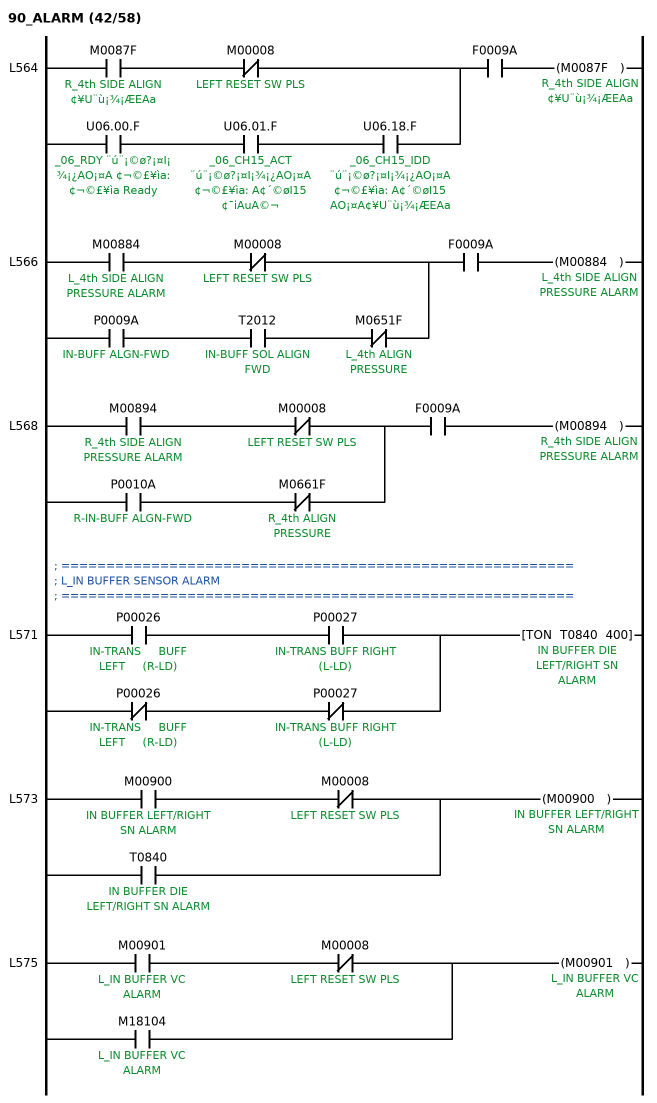
[picture p408: 90_ALARM rungs L564-L575]
; L564
LOAD      M0087F	// R_4th SIDE ALIGN ¢¥U¨ù¡¾¡ÆEAa
AND NOT   M00008	// LEFT RESET SW PLS
LOAD      U06.00.F	// _06_RDY ¨ú¨¡©ø?¡¤I¡¾¡¿AO¡¤A ¢¬©£¥ìa: ¢¬©£¥ìa Ready
AND       U06.01.F	// _06_CH15_ACT ¨ú¨¡©ø?¡¤I¡¾¡¿AO¡¤A ¢¬©£¥ìa: A¢´©øI15 ¢¯iAuA©¬
AND       U06.18.F	// _06_CH15_IDD ¨ú¨¡©ø?¡¤I¡¾¡¿AO¡¤A ¢¬©£¥ìa: A¢´©øI15 AO¡¤A¢¥U¨ù¡¾¡ÆEAa
OR LOAD
AND       F0009A
OUT       M0087F	// R_4th SIDE ALIGN ¢¥U¨ù¡¾¡ÆEAa
; L566
LOAD      M00884	// L_4th SIDE ALIGN PRESSURE ALARM
AND NOT   M00008	// LEFT RESET SW PLS
LOAD      P0009A	// IN-BUFF ALGN-FWD
AND       T2012	// IN-BUFF SOL ALIGN FWD
AND NOT   M0651F	// L_4th ALIGN PRESSURE
OR LOAD
AND       F0009A
OUT       M00884	// L_4th SIDE ALIGN PRESSURE ALARM
; L568
LOAD      M00894	// R_4th SIDE ALIGN PRESSURE ALARM
AND NOT   M00008	// LEFT RESET SW PLS
LOAD      P0010A	// R-IN-BUFF ALGN-FWD
AND NOT   M0661F	// R_4th ALIGN PRESSURE
OR LOAD
AND       F0009A
OUT       M00894	// R_4th SIDE ALIGN PRESSURE ALARM
// =========================================================
// 
//        L_IN BUFFER SENSOR ALARM
// 
// =========================================================
; L571
LOAD      P00026	// IN-TRANS     BUFF     LEFT     (R-LD)
AND       P00027	// IN-TRANS BUFF RIGHT     (L-LD)
LOAD NOT  P00026	// IN-TRANS     BUFF     LEFT     (R-LD)
AND NOT   P00027	// IN-TRANS BUFF RIGHT     (L-LD)
OR LOAD
TON       T0840 400	// IN BUFFER DIE LEFT/RIGHT SN ALARM
; L573
LOAD      M00900	// IN BUFFER LEFT/RIGHT SN ALARM
AND NOT   M00008	// LEFT RESET SW PLS
OR        T0840	// IN BUFFER DIE LEFT/RIGHT SN ALARM
OUT       M00900	// IN BUFFER LEFT/RIGHT SN ALARM
; L575
LOAD      M00901	// L_IN BUFFER VC ALARM
AND NOT   M00008	// LEFT RESET SW PLS
OR        M18104	// L_IN BUFFER VC ALARM
OUT       M00901	// L_IN BUFFER VC ALARM

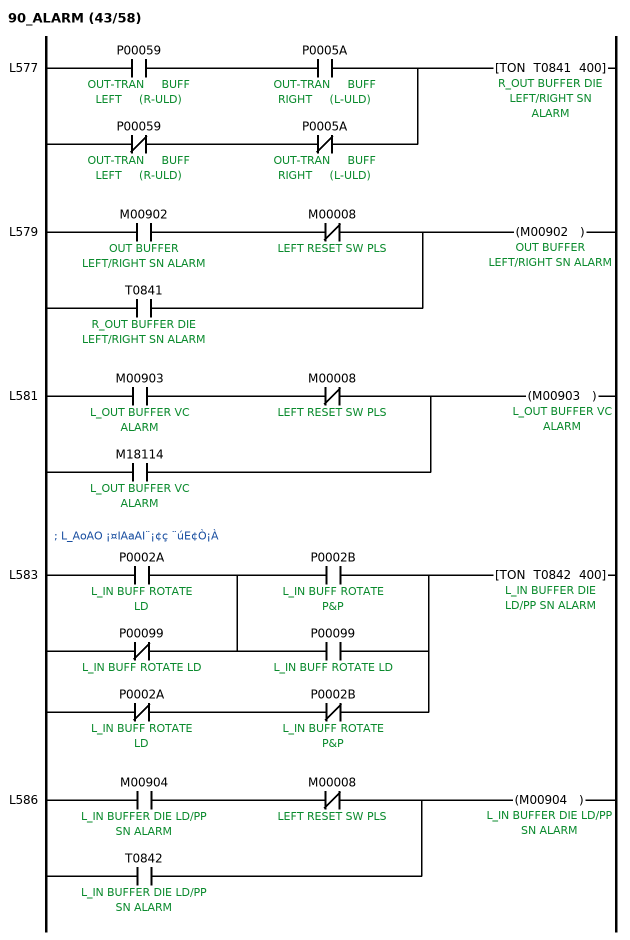
; L577
LOAD      P00059	// OUT-TRAN     BUFF     LEFT     (R-ULD)
AND       P0005A	// OUT-TRAN     BUFF     RIGHT     (L-ULD)
LOAD NOT  P00059	// OUT-TRAN     BUFF     LEFT     (R-ULD)
AND NOT   P0005A	// OUT-TRAN     BUFF     RIGHT     (L-ULD)
OR LOAD
TON       T0841 400	// R_OUT BUFFER DIE LEFT/RIGHT SN ALARM
; L579
LOAD      M00902	// OUT BUFFER LEFT/RIGHT SN ALARM
AND NOT   M00008	// LEFT RESET SW PLS
OR        T0841	// R_OUT BUFFER DIE LEFT/RIGHT SN ALARM
OUT       M00902	// OUT BUFFER LEFT/RIGHT SN ALARM
; L581
LOAD      M00903	// L_OUT BUFFER VC ALARM
AND NOT   M00008	// LEFT RESET SW PLS
OR        M18114	// L_OUT BUFFER VC ALARM
OUT       M00903	// L_OUT BUFFER VC ALARM
; L583
LOAD      P0002A	// L_IN BUFF ROTATE     LD
OR NOT    P00099	// L_IN BUFF ROTATE LD
LOAD      P0002B	// L_IN BUFF ROTATE      P&P
OR        P00099	// L_IN BUFF ROTATE LD
AND LOAD
LOAD NOT  P0002A	// L_IN BUFF ROTATE     LD
AND NOT   P0002B	// L_IN BUFF ROTATE      P&P
OR LOAD
TON       T0842 400	// L_IN BUFFER DIE LD/PP SN ALARM
// output comment: L_AoAO ¡¤IAaAI¨¡¢ç ¨úE¢Ò¡À
; L586
LOAD      M00904	// L_IN BUFFER DIE LD/PP SN ALARM
AND NOT   M00008	// LEFT RESET SW PLS
OR        T0842	// L_IN BUFFER DIE LD/PP SN ALARM
OUT       M00904	// L_IN BUFFER DIE LD/PP SN ALARM

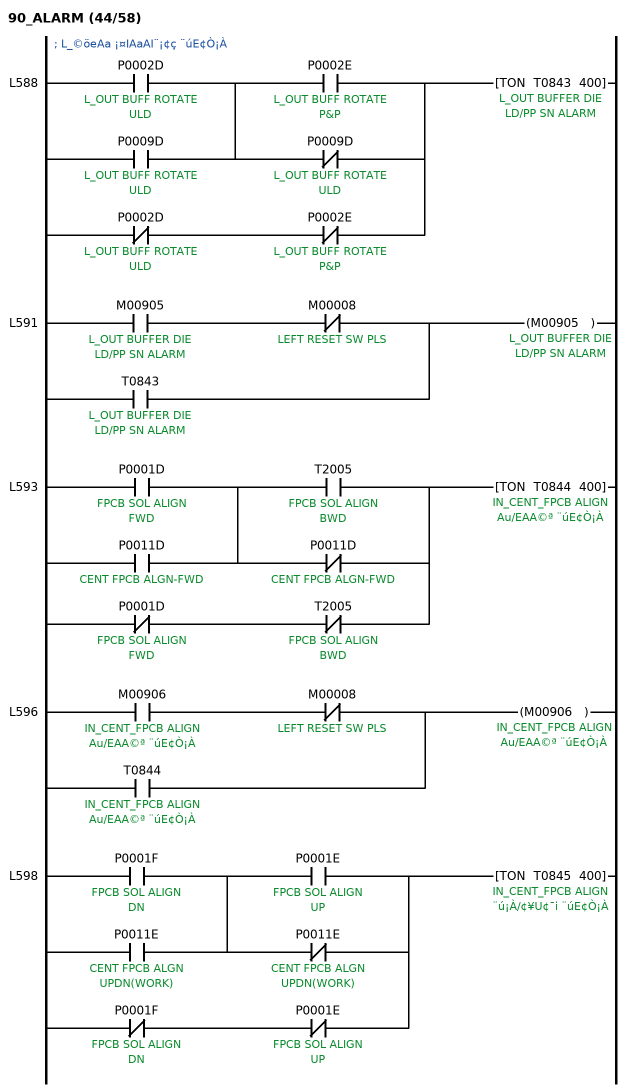
; L588
LOAD      P0002D	// L_OUT BUFF ROTATE     ULD
OR        P0009D	// L_OUT BUFF ROTATE ULD
LOAD      P0002E	// L_OUT BUFF ROTATE      P&P
OR NOT    P0009D	// L_OUT BUFF ROTATE ULD
AND LOAD
LOAD NOT  P0002D	// L_OUT BUFF ROTATE     ULD
AND NOT   P0002E	// L_OUT BUFF ROTATE      P&P
OR LOAD
TON       T0843 400	// L_OUT BUFFER DIE LD/PP SN ALARM
// output comment: L_©öeAa ¡¤IAaAI¨¡¢ç ¨úE¢Ò¡À
; L591
LOAD      M00905	// L_OUT BUFFER DIE LD/PP SN ALARM
AND NOT   M00008	// LEFT RESET SW PLS
OR        T0843	// L_OUT BUFFER DIE LD/PP SN ALARM
OUT       M00905	// L_OUT BUFFER DIE LD/PP SN ALARM
; L593
LOAD      P0001D	// FPCB SOL ALIGN         FWD
OR        P0011D	// CENT FPCB ALGN-FWD
LOAD      T2005	// FPCB SOL ALIGN         BWD
OR NOT    P0011D	// CENT FPCB ALGN-FWD
AND LOAD
LOAD NOT  P0001D	// FPCB SOL ALIGN         FWD
AND NOT   T2005	// FPCB SOL ALIGN         BWD
OR LOAD
TON       T0844 400	// IN_CENT_FPCB ALIGN Au/EAA©ª ¨úE¢Ò¡À
; L596
LOAD      M00906	// IN_CENT_FPCB ALIGN Au/EAA©ª ¨úE¢Ò¡À
AND NOT   M00008	// LEFT RESET SW PLS
OR        T0844	// IN_CENT_FPCB ALIGN Au/EAA©ª ¨úE¢Ò¡À
OUT       M00906	// IN_CENT_FPCB ALIGN Au/EAA©ª ¨úE¢Ò¡À
; L598
LOAD      P0001F	// FPCB SOL ALIGN        DN
OR        P0011E	// CENT FPCB ALGN UPDN(WORK)
LOAD      P0001E	// FPCB SOL ALIGN         UP
OR NOT    P0011E	// CENT FPCB ALGN UPDN(WORK)
AND LOAD
LOAD NOT  P0001F	// FPCB SOL ALIGN        DN
AND NOT   P0001E	// FPCB SOL ALIGN         UP
OR LOAD
TON       T0845 400	// IN_CENT_FPCB ALIGN ¨ú¡À/¢¥U¢¯i ¨úE¢Ò¡À

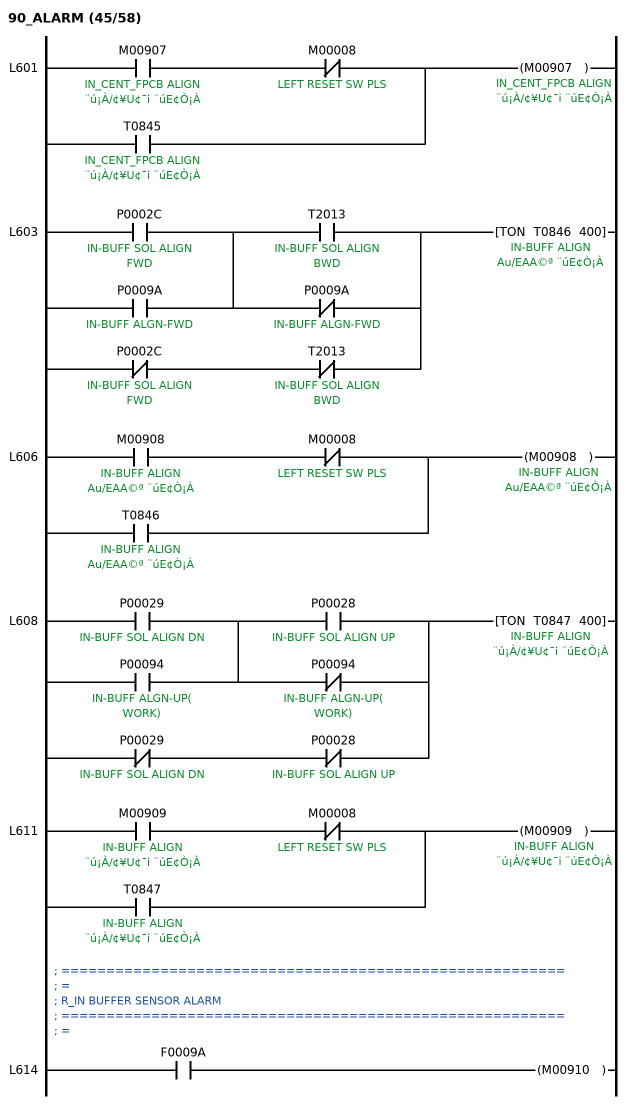
; L601
LOAD      M00907	// IN_CENT_FPCB ALIGN ¨ú¡À/¢¥U¢¯i ¨úE¢Ò¡À
AND NOT   M00008	// LEFT RESET SW PLS
OR        T0845	// IN_CENT_FPCB ALIGN ¨ú¡À/¢¥U¢¯i ¨úE¢Ò¡À
OUT       M00907	// IN_CENT_FPCB ALIGN ¨ú¡À/¢¥U¢¯i ¨úE¢Ò¡À
; L603
LOAD      P0002C	// IN-BUFF SOL ALIGN FWD
OR        P0009A	// IN-BUFF ALGN-FWD
LOAD      T2013	// IN-BUFF SOL ALIGN BWD
OR NOT    P0009A	// IN-BUFF ALGN-FWD
AND LOAD
LOAD NOT  P0002C	// IN-BUFF SOL ALIGN FWD
AND NOT   T2013	// IN-BUFF SOL ALIGN BWD
OR LOAD
TON       T0846 400	// IN-BUFF ALIGN Au/EAA©ª ¨úE¢Ò¡À
; L606
LOAD      M00908	// IN-BUFF ALIGN Au/EAA©ª ¨úE¢Ò¡À
AND NOT   M00008	// LEFT RESET SW PLS
OR        T0846	// IN-BUFF ALIGN Au/EAA©ª ¨úE¢Ò¡À
OUT       M00908	// IN-BUFF ALIGN Au/EAA©ª ¨úE¢Ò¡À
; L608
LOAD      P00029	// IN-BUFF SOL ALIGN DN
OR        P00094	// IN-BUFF ALGN-UP(WORK)
LOAD      P00028	// IN-BUFF SOL ALIGN UP
OR NOT    P00094	// IN-BUFF ALGN-UP(WORK)
AND LOAD
LOAD NOT  P00029	// IN-BUFF SOL ALIGN DN
AND NOT   P00028	// IN-BUFF SOL ALIGN UP
OR LOAD
TON       T0847 400	// IN-BUFF ALIGN ¨ú¡À/¢¥U¢¯i ¨úE¢Ò¡À
; L611
LOAD      M00909	// IN-BUFF ALIGN ¨ú¡À/¢¥U¢¯i ¨úE¢Ò¡À
AND NOT   M00008	// LEFT RESET SW PLS
OR        T0847	// IN-BUFF ALIGN ¨ú¡À/¢¥U¢¯i ¨úE¢Ò¡À
OUT       M00909	// IN-BUFF ALIGN ¨ú¡À/¢¥U¢¯i ¨úE¢Ò¡À
// =========================================================
// 
//        R_IN BUFFER SENSOR ALARM
// 
// =========================================================
; L614
LOAD      F0009A
OUT       M00910

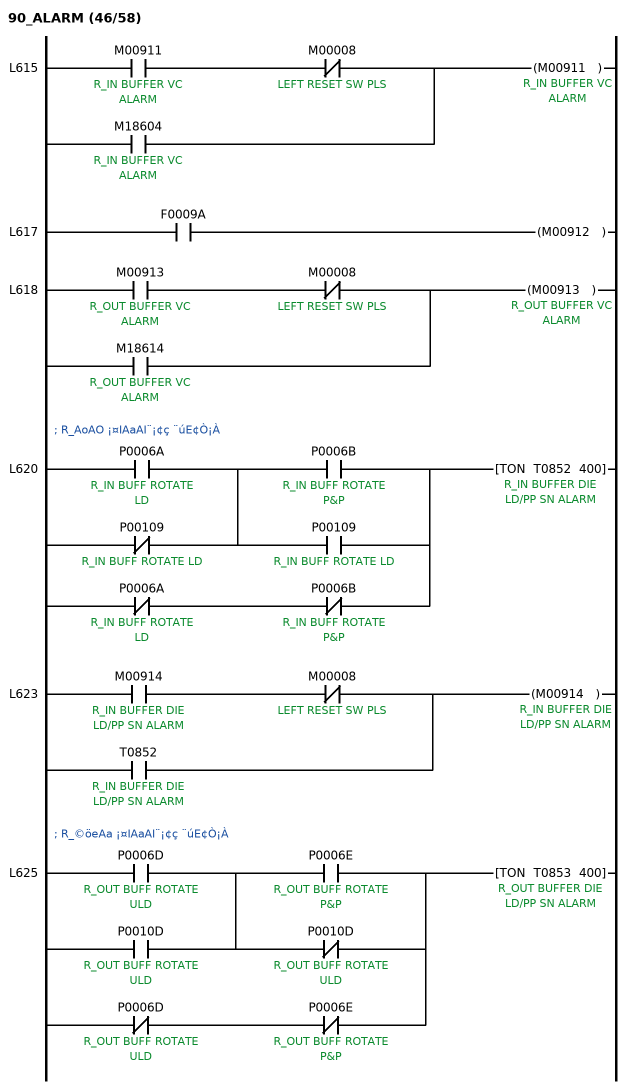
; L615
LOAD      M00911	// R_IN BUFFER VC ALARM
AND NOT   M00008	// LEFT RESET SW PLS
OR        M18604	// R_IN BUFFER VC ALARM
OUT       M00911	// R_IN BUFFER VC ALARM
; L617
LOAD      F0009A
OUT       M00912
; L618
LOAD      M00913	// R_OUT BUFFER VC ALARM
AND NOT   M00008	// LEFT RESET SW PLS
OR        M18614	// R_OUT BUFFER VC ALARM
OUT       M00913	// R_OUT BUFFER VC ALARM
; L620
LOAD      P0006A	// R_IN BUFF ROTATE      LD
OR NOT    P00109	// R_IN BUFF ROTATE LD
LOAD      P0006B	// R_IN BUFF ROTATE      P&P
OR        P00109	// R_IN BUFF ROTATE LD
AND LOAD
LOAD NOT  P0006A	// R_IN BUFF ROTATE      LD
AND NOT   P0006B	// R_IN BUFF ROTATE      P&P
OR LOAD
TON       T0852 400	// R_IN BUFFER DIE LD/PP SN ALARM
// output comment: R_AoAO ¡¤IAaAI¨¡¢ç ¨úE¢Ò¡À
; L623
LOAD      M00914	// R_IN BUFFER DIE LD/PP SN ALARM
AND NOT   M00008	// LEFT RESET SW PLS
OR        T0852	// R_IN BUFFER DIE LD/PP SN ALARM
OUT       M00914	// R_IN BUFFER DIE LD/PP SN ALARM
; L625
LOAD      P0006D	// R_OUT BUFF ROTATE      ULD
OR        P0010D	// R_OUT BUFF ROTATE ULD
LOAD      P0006E	// R_OUT BUFF ROTATE      P&P
OR NOT    P0010D	// R_OUT BUFF ROTATE ULD
AND LOAD
LOAD NOT  P0006D	// R_OUT BUFF ROTATE      ULD
AND NOT   P0006E	// R_OUT BUFF ROTATE      P&P
OR LOAD
TON       T0853 400	// R_OUT BUFFER DIE LD/PP SN ALARM
// output comment: R_©öeAa ¡¤IAaAI¨¡¢ç ¨úE¢Ò¡À

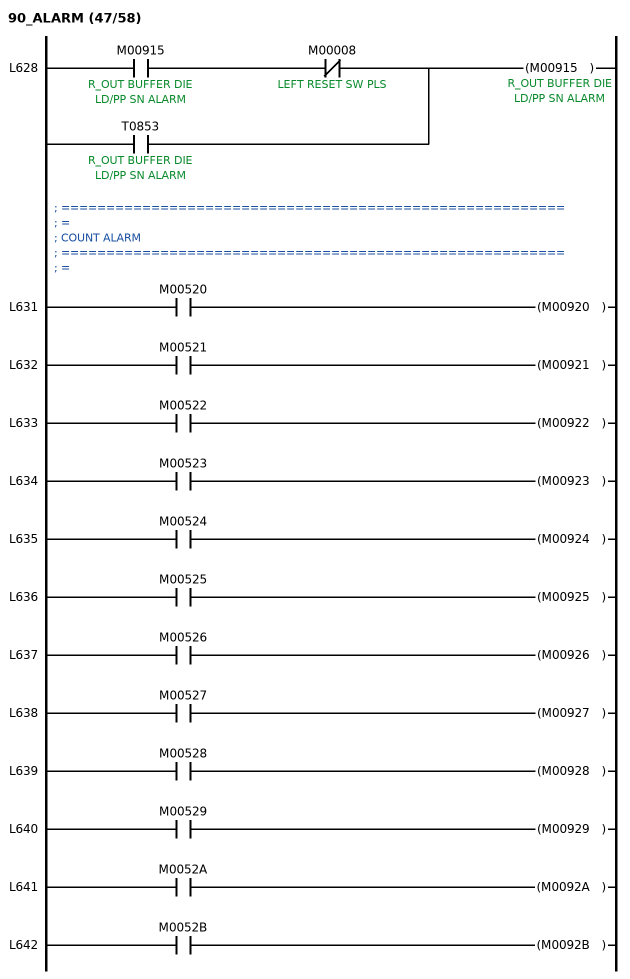
; L628
LOAD      M00915	// R_OUT BUFFER DIE LD/PP SN ALARM
AND NOT   M00008	// LEFT RESET SW PLS
OR        T0853	// R_OUT BUFFER DIE LD/PP SN ALARM
OUT       M00915	// R_OUT BUFFER DIE LD/PP SN ALARM
// =========================================================
// 
//       COUNT ALARM
// 
// =========================================================
; L631
LOAD      M00520
OUT       M00920
; L632
LOAD      M00521
OUT       M00921
; L633
LOAD      M00522
OUT       M00922
; L634
LOAD      M00523
OUT       M00923
; L635
LOAD      M00524
OUT       M00924
; L636
LOAD      M00525
OUT       M00925
; L637
LOAD      M00526
OUT       M00926
; L638
LOAD      M00527
OUT       M00927
; L639
LOAD      M00528
OUT       M00928
; L640
LOAD      M00529
OUT       M00929
; L641
LOAD      M0052A
OUT       M0092A
; L642
LOAD      M0052B
OUT       M0092B

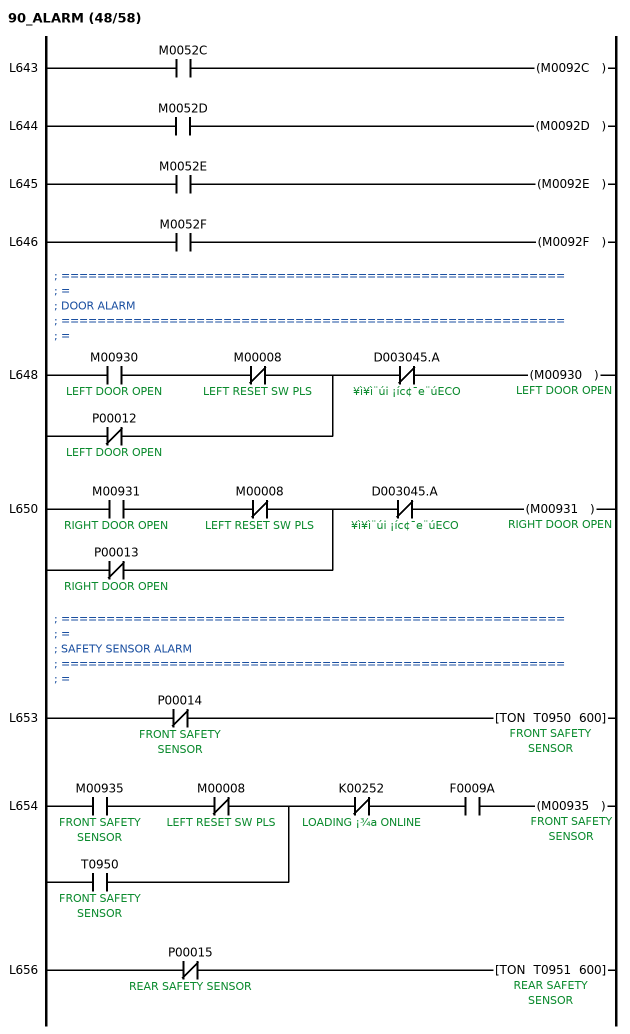
; L643
LOAD      M0052C
OUT       M0092C
; L644
LOAD      M0052D
OUT       M0092D
; L645
LOAD      M0052E
OUT       M0092E
; L646
LOAD      M0052F
OUT       M0092F
// =========================================================
// 
//       DOOR ALARM
// 
// =========================================================
; L648
LOAD      M00930	// LEFT DOOR OPEN
AND NOT   M00008	// LEFT RESET SW PLS
OR NOT    P00012	// LEFT DOOR OPEN
AND NOT   D003045.A	// ¥ì¥ì¨úi ¡íc¢¯e¨úECO
OUT       M00930	// LEFT DOOR OPEN
; L650
LOAD      M00931	// RIGHT DOOR OPEN
AND NOT   M00008	// LEFT RESET SW PLS
OR NOT    P00013	// RIGHT DOOR OPEN
AND NOT   D003045.A	// ¥ì¥ì¨úi ¡íc¢¯e¨úECO
OUT       M00931	// RIGHT DOOR OPEN
// =========================================================
// 
//       SAFETY SENSOR ALARM
// 
// =========================================================
; L653
LOAD NOT  P00014	// FRONT SAFETY SENSOR
TON       T0950 600	// FRONT SAFETY SENSOR
; L654
LOAD      M00935	// FRONT SAFETY SENSOR
AND NOT   M00008	// LEFT RESET SW PLS
OR        T0950	// FRONT SAFETY SENSOR
AND NOT   K00252	// LOADING ¡¾a ONLINE
AND       F0009A
OUT       M00935	// FRONT SAFETY SENSOR
; L656
LOAD NOT  P00015	// REAR SAFETY SENSOR
TON       T0951 600	// REAR SAFETY SENSOR

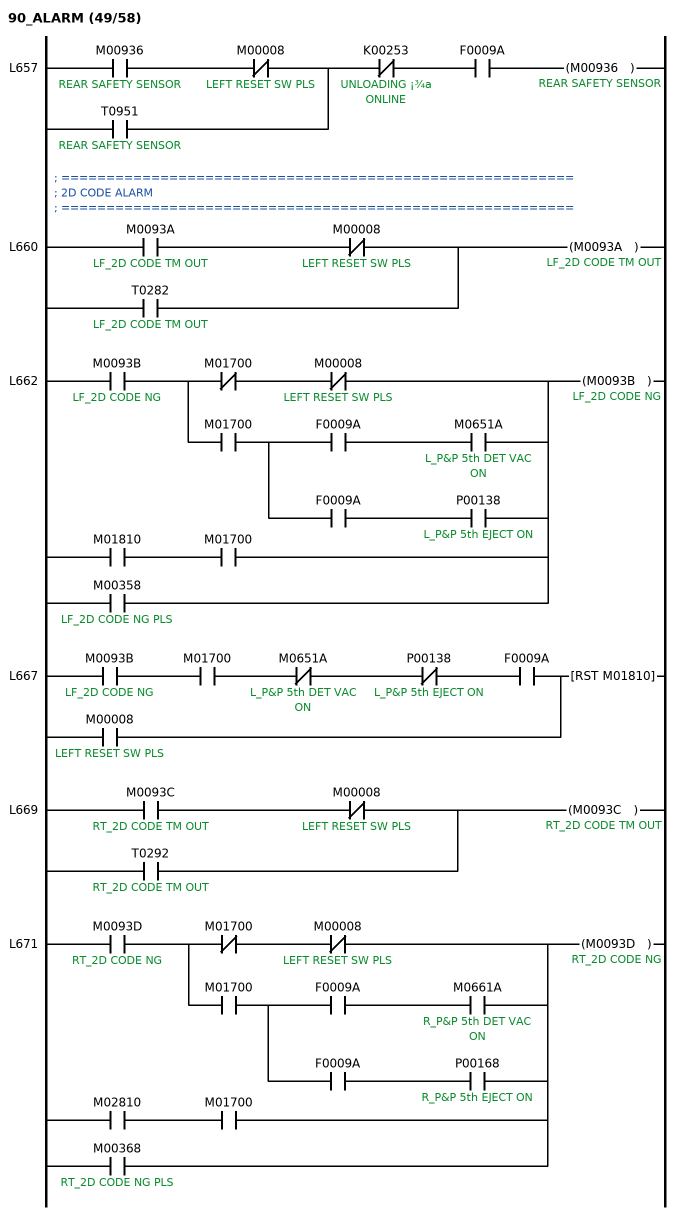
; L657
LOAD      M00936	// REAR SAFETY SENSOR
AND NOT   M00008	// LEFT RESET SW PLS
OR        T0951	// REAR SAFETY SENSOR
AND NOT   K00253	// UNLOADING ¡¾a ONLINE
AND       F0009A
OUT       M00936	// REAR SAFETY SENSOR
// =========================================================
// 
//       2D CODE ALARM
// 
// =========================================================
; L660
LOAD      M0093A	// LF_2D CODE TM OUT
AND NOT   M00008	// LEFT RESET SW PLS
OR        T0282	// LF_2D CODE TM OUT
OUT       M0093A	// LF_2D CODE TM OUT
; L662
LOAD      M0093B	// LF_2D CODE NG
LOAD NOT  M01700
AND NOT   M00008	// LEFT RESET SW PLS
LOAD      M01700
LOAD      F0009A
AND       M0651A	// L_P&P 5th DET VAC ON
LOAD      F0009A
AND       P00138	// L_P&P 5th EJECT ON
OR LOAD
AND LOAD
OR LOAD
AND LOAD
LOAD      M01810
AND       M01700
OR LOAD
OR        M00358	// LF_2D CODE NG PLS
OUT       M0093B	// LF_2D CODE NG
; L667
LOAD      M0093B	// LF_2D CODE NG
AND       M01700
AND NOT   M0651A	// L_P&P 5th DET VAC ON
AND NOT   P00138	// L_P&P 5th EJECT ON
AND       F0009A
OR        M00008	// LEFT RESET SW PLS
RST       M01810
; L669
LOAD      M0093C	// RT_2D CODE TM OUT
AND NOT   M00008	// LEFT RESET SW PLS
OR        T0292	// RT_2D CODE TM OUT
OUT       M0093C	// RT_2D CODE TM OUT
; L671
LOAD      M0093D	// RT_2D CODE NG
LOAD NOT  M01700
AND NOT   M00008	// LEFT RESET SW PLS
LOAD      M01700
LOAD      F0009A
AND       M0661A	// R_P&P 5th DET VAC ON
LOAD      F0009A
AND       P00168	// R_P&P 5th EJECT ON
OR LOAD
AND LOAD
OR LOAD
AND LOAD
LOAD      M02810
AND       M01700
OR LOAD
OR        M00368	// RT_2D CODE NG PLS
OUT       M0093D	// RT_2D CODE NG

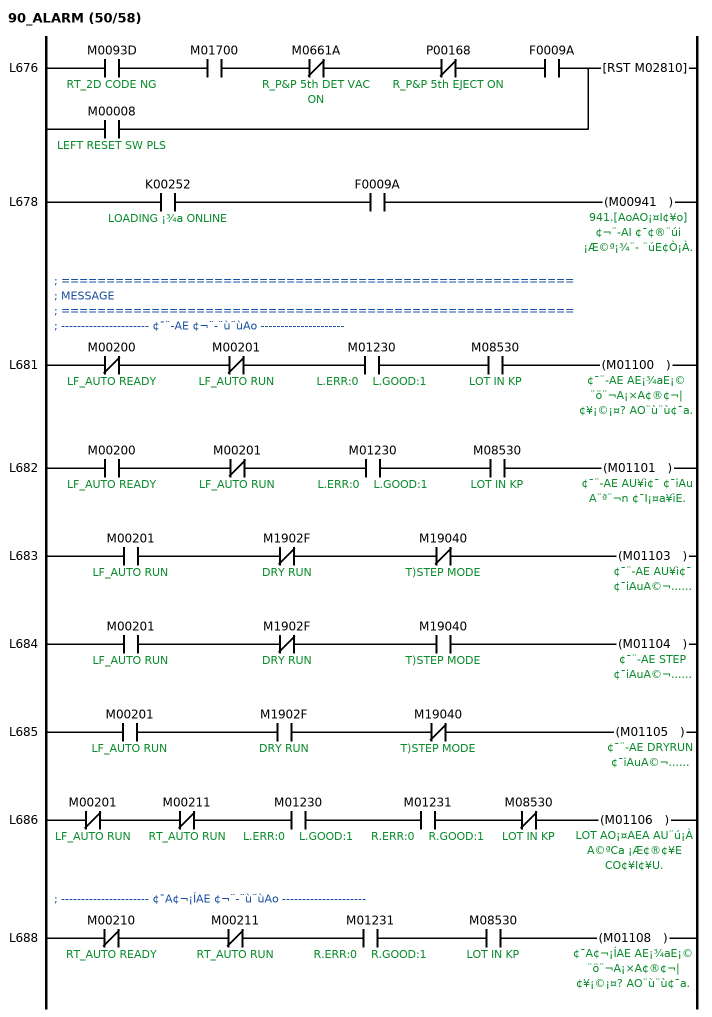
; L676
LOAD      M0093D	// RT_2D CODE NG
AND       M01700
AND NOT   M0661A	// R_P&P 5th DET VAC ON
AND NOT   P00168	// R_P&P 5th EJECT ON
AND       F0009A
OR        M00008	// LEFT RESET SW PLS
RST       M02810
; L678
LOAD      K00252	// LOADING ¡¾a ONLINE
AND       F0009A
OUT       M00941	// 941.[AoAO¡¤I¢¥o] ¢¬¨­AI ¢¯¢®¨úi ¡Æ©ª¡¾¨­ ¨úE¢Ò¡À.
// =========================================================
// 
//       MESSAGE
// 
// =========================================================
// ---------------------- ¢¯¨­AE ¢¬¨­¨ù¨ùAo ---------------------
; L681
LOAD NOT  M00200	// LF_AUTO READY
AND NOT   M00201	// LF_AUTO RUN
AND       M01230	// L.ERR:0    L.GOOD:1
AND       M08530	// LOT IN KP
OUT       M01100	// ¢¯¨­AE AE¡¾aE¡© ¨ö¨¬A¡×A¢®¢¬| ¢¥¡©¡¤? AO¨ù¨ù¢¯a.
; L682
LOAD      M00200	// LF_AUTO READY
AND NOT   M00201	// LF_AUTO RUN
AND       M01230	// L.ERR:0    L.GOOD:1
AND       M08530	// LOT IN KP
OUT       M01101	// ¢¯¨­AE AU¥ì¢¯ ¢¯iAu A¨ª¨¬n ¢¯I¡¤a¥ìE.
; L683
LOAD      M00201	// LF_AUTO RUN
AND NOT   M1902F	// DRY RUN
AND NOT   M19040	// T)STEP MODE
OUT       M01103	// ¢¯¨­AE AU¥ì¢¯ ¢¯iAuA©¬......
; L684
LOAD      M00201	// LF_AUTO RUN
AND NOT   M1902F	// DRY RUN
AND       M19040	// T)STEP MODE
OUT       M01104	// ¢¯¨­AE STEP ¢¯iAuA©¬......
; L685
LOAD      M00201	// LF_AUTO RUN
AND       M1902F	// DRY RUN
AND NOT   M19040	// T)STEP MODE
OUT       M01105	// ¢¯¨­AE DRYRUN ¢¯iAuA©¬......
; L686
LOAD NOT  M00201	// LF_AUTO RUN
AND NOT   M00211	// RT_AUTO RUN
AND       M01230	// L.ERR:0    L.GOOD:1
AND       M01231	// R.ERR:0    R.GOOD:1
AND NOT   M08530	// LOT IN KP
OUT       M01106	// LOT AO¡¤AEA AU¨ú¡À A©ªCa ¡Æ¢®¢¥E CO¢¥I¢¥U.
// ---------------------- ¢¯A¢¬¡ÍAE ¢¬¨­¨ù¨ùAo ---------------------
; L688
LOAD NOT  M00210	// RT_AUTO READY
AND NOT   M00211	// RT_AUTO RUN
AND       M01231	// R.ERR:0    R.GOOD:1
AND       M08530	// LOT IN KP
OUT       M01108	// ¢¯A¢¬¡ÍAE AE¡¾aE¡© ¨ö¨¬A¡×A¢®¢¬| ¢¥¡©¡¤? AO¨ù¨ù¢¯a.

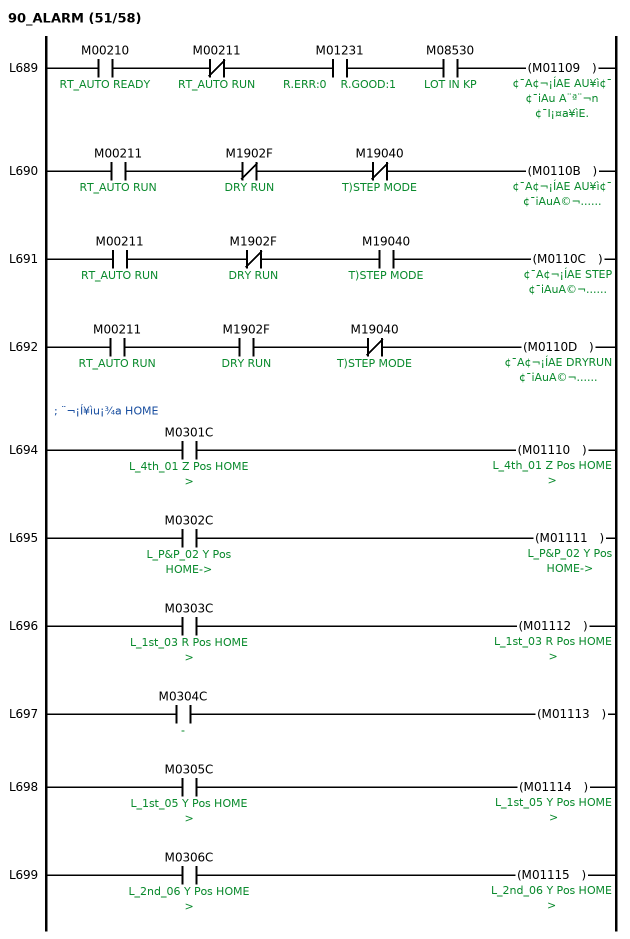
; L689
LOAD      M00210	// RT_AUTO READY
AND NOT   M00211	// RT_AUTO RUN
AND       M01231	// R.ERR:0    R.GOOD:1
AND       M08530	// LOT IN KP
OUT       M01109	// ¢¯A¢¬¡ÍAE AU¥ì¢¯ ¢¯iAu A¨ª¨¬n ¢¯I¡¤a¥ìE.
; L690
LOAD      M00211	// RT_AUTO RUN
AND NOT   M1902F	// DRY RUN
AND NOT   M19040	// T)STEP MODE
OUT       M0110B	// ¢¯A¢¬¡ÍAE AU¥ì¢¯ ¢¯iAuA©¬......
; L691
LOAD      M00211	// RT_AUTO RUN
AND NOT   M1902F	// DRY RUN
AND       M19040	// T)STEP MODE
OUT       M0110C	// ¢¯A¢¬¡ÍAE STEP ¢¯iAuA©¬......
; L692
LOAD      M00211	// RT_AUTO RUN
AND       M1902F	// DRY RUN
AND NOT   M19040	// T)STEP MODE
OUT       M0110D	// ¢¯A¢¬¡ÍAE DRYRUN ¢¯iAuA©¬......
// ¨¬¡Í¥ìu¡¾a HOME
; L694
LOAD      M0301C	// L_4th_01 Z Pos HOME >
OUT       M01110	// L_4th_01 Z Pos HOME >
; L695
LOAD      M0302C	// L_P&P_02 Y Pos HOME->
OUT       M01111	// L_P&P_02 Y Pos HOME->
; L696
LOAD      M0303C	// L_1st_03 R Pos HOME >
OUT       M01112	// L_1st_03 R Pos HOME >
; L697
LOAD      M0304C	// -
OUT       M01113
; L698
LOAD      M0305C	// L_1st_05 Y Pos HOME >
OUT       M01114	// L_1st_05 Y Pos HOME >
; L699
LOAD      M0306C	// L_2nd_06 Y Pos HOME >
OUT       M01115	// L_2nd_06 Y Pos HOME >

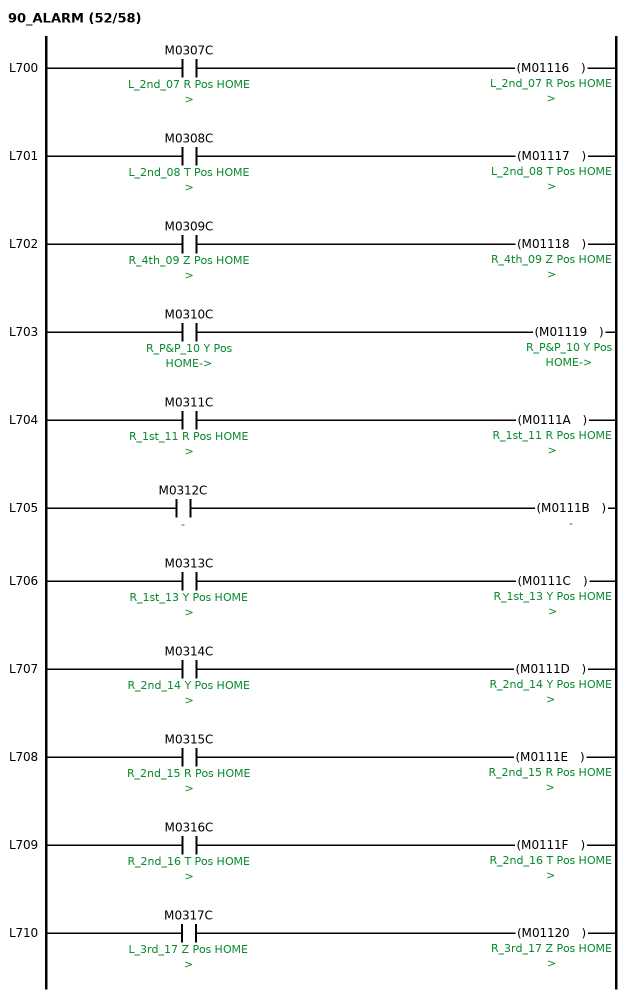
; L700
LOAD      M0307C	// L_2nd_07 R Pos HOME >
OUT       M01116	// L_2nd_07 R Pos HOME >
; L701
LOAD      M0308C	// L_2nd_08 T Pos HOME >
OUT       M01117	// L_2nd_08 T Pos HOME >
; L702
LOAD      M0309C	// R_4th_09 Z Pos HOME >
OUT       M01118	// R_4th_09 Z Pos HOME >
; L703
LOAD      M0310C	// R_P&P_10 Y Pos HOME->
OUT       M01119	// R_P&P_10 Y Pos HOME->
; L704
LOAD      M0311C	// R_1st_11 R Pos HOME >
OUT       M0111A	// R_1st_11 R Pos HOME >
; L705
LOAD      M0312C	// -
OUT       M0111B	// -
; L706
LOAD      M0313C	// R_1st_13 Y Pos HOME >
OUT       M0111C	// R_1st_13 Y Pos HOME >
; L707
LOAD      M0314C	// R_2nd_14 Y Pos HOME >
OUT       M0111D	// R_2nd_14 Y Pos HOME >
; L708
LOAD      M0315C	// R_2nd_15 R Pos HOME >
OUT       M0111E	// R_2nd_15 R Pos HOME >
; L709
LOAD      M0316C	// R_2nd_16 T Pos HOME >
OUT       M0111F	// R_2nd_16 T Pos HOME >
; L710
LOAD      M0317C	// L_3rd_17 Z Pos HOME >
OUT       M01120	// R_3rd_17 Z Pos HOME >

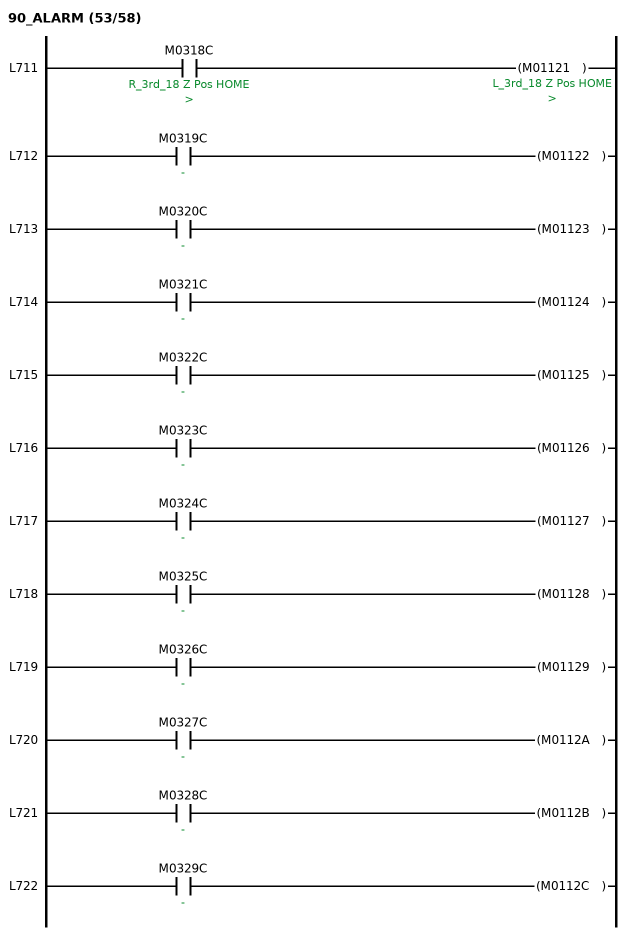
; L711
LOAD      M0318C	// R_3rd_18 Z Pos HOME >
OUT       M01121	// L_3rd_18 Z Pos HOME >
; L712
LOAD      M0319C	// -
OUT       M01122
; L713
LOAD      M0320C	// -
OUT       M01123
; L714
LOAD      M0321C	// -
OUT       M01124
; L715
LOAD      M0322C	// -
OUT       M01125
; L716
LOAD      M0323C	// -
OUT       M01126
; L717
LOAD      M0324C	// -
OUT       M01127
; L718
LOAD      M0325C	// -
OUT       M01128
; L719
LOAD      M0326C	// -
OUT       M01129
; L720
LOAD      M0327C	// -
OUT       M0112A
; L721
LOAD      M0328C	// -
OUT       M0112B
; L722
LOAD      M0329C	// -
OUT       M0112C

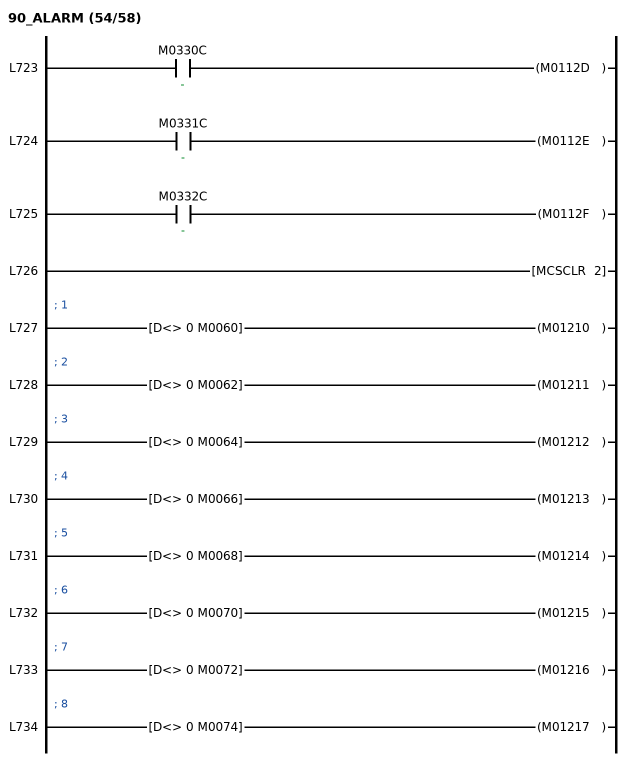
; L723
LOAD      M0330C	// -
OUT       M0112D
; L724
LOAD      M0331C	// -
OUT       M0112E
; L725
LOAD      M0332C	// -
OUT       M0112F
; L726
MCSCLR    2
; L727
LOADD<>   0 M0060
OUT       M01210
// output comment: 1
; L728
LOADD<>   0 M0062
OUT       M01211
// output comment: 2
; L729
LOADD<>   0 M0064
OUT       M01212
// output comment: 3
; L730
LOADD<>   0 M0066
OUT       M01213
// output comment: 4
; L731
LOADD<>   0 M0068
OUT       M01214
// output comment: 5
; L732
LOADD<>   0 M0070
OUT       M01215
// output comment: 6
; L733
LOADD<>   0 M0072
OUT       M01216
// output comment: 7
; L734
LOADD<>   0 M0074
OUT       M01217
// output comment: 8

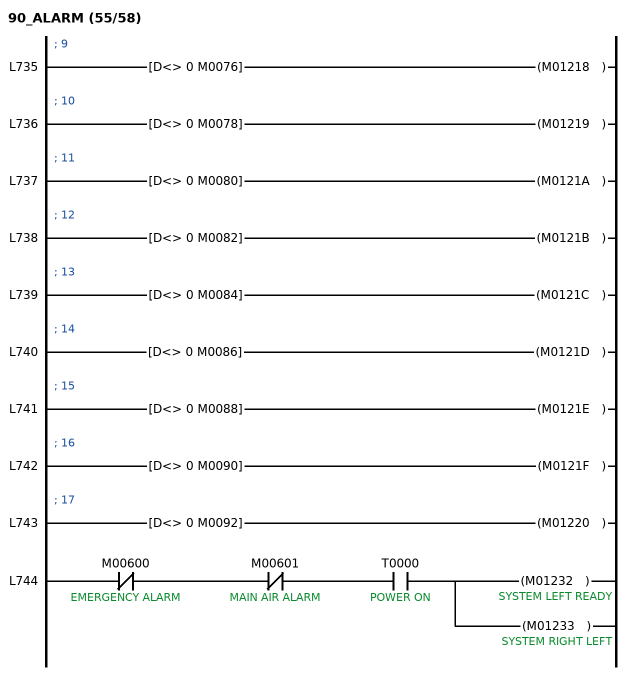
; L735
LOADD<>   0 M0076
OUT       M01218
// output comment: 9
; L736
LOADD<>   0 M0078
OUT       M01219
// output comment: 10
; L737
LOADD<>   0 M0080
OUT       M0121A
// output comment: 11
; L738
LOADD<>   0 M0082
OUT       M0121B
// output comment: 12
; L739
LOADD<>   0 M0084
OUT       M0121C
// output comment: 13
; L740
LOADD<>   0 M0086
OUT       M0121D
// output comment: 14
; L741
LOADD<>   0 M0088
OUT       M0121E
// output comment: 15
; L742
LOADD<>   0 M0090
OUT       M0121F
// output comment: 16
; L743
LOADD<>   0 M0092
OUT       M01220
// output comment: 17
; L744
LOAD NOT  M00600	// EMERGENCY ALARM
AND NOT   M00601	// MAIN AIR ALARM
AND       T0000	// POWER ON
OUT       M01232	// SYSTEM LEFT READY
OUT       M01233	// SYSTEM RIGHT LEFT

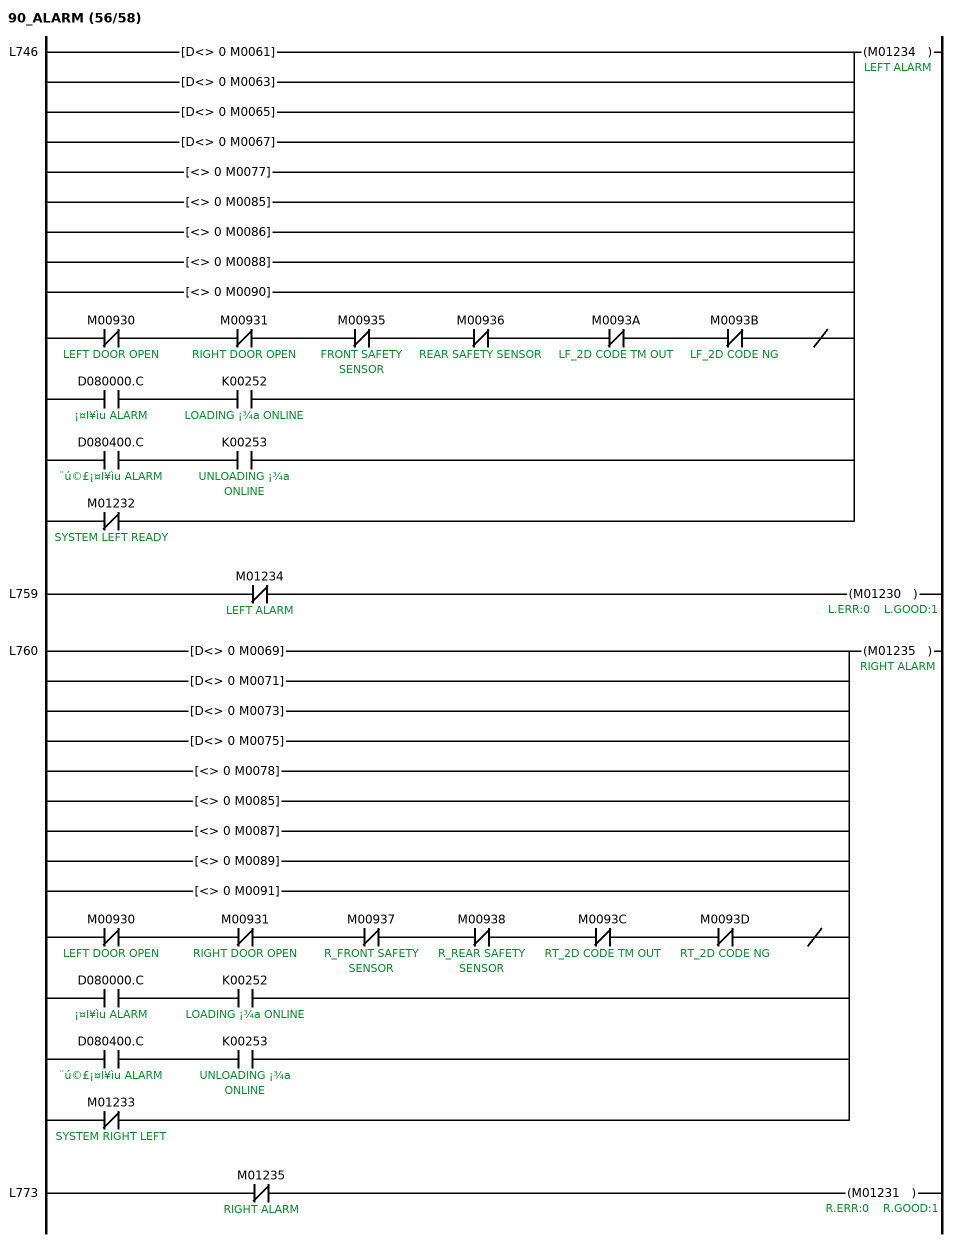
; L746
LOADD<>   0 M0061
ORD<>     0 M0063
ORD<>     0 M0065
ORD<>     0 M0067
OR<>      0 M0077
OR<>      0 M0085
OR<>      0 M0086
OR<>      0 M0088
OR<>      0 M0090
LOAD NOT  M00930	// LEFT DOOR OPEN
AND NOT   M00931	// RIGHT DOOR OPEN
AND NOT   M00935	// FRONT SAFETY SENSOR
AND NOT   M00936	// REAR SAFETY SENSOR
AND NOT   M0093A	// LF_2D CODE TM OUT
AND NOT   M0093B	// LF_2D CODE NG
NOT
OR LOAD
LOAD      D080000.C	// ¡¤I¥ìu ALARM
AND       K00252	// LOADING ¡¾a ONLINE
OR LOAD
LOAD      D080400.C	// ¨ú©£¡¤I¥ìu ALARM
AND       K00253	// UNLOADING ¡¾a ONLINE
OR LOAD
OR NOT    M01232	// SYSTEM LEFT READY
OUT       M01234	// LEFT ALARM
; L759
LOAD NOT  M01234	// LEFT ALARM
OUT       M01230	// L.ERR:0    L.GOOD:1
; L760
LOADD<>   0 M0069
ORD<>     0 M0071
ORD<>     0 M0073
ORD<>     0 M0075
OR<>      0 M0078
OR<>      0 M0085
OR<>      0 M0087
OR<>      0 M0089
OR<>      0 M0091
LOAD NOT  M00930	// LEFT DOOR OPEN
AND NOT   M00931	// RIGHT DOOR OPEN
AND NOT   M00937	// R_FRONT SAFETY SENSOR
AND NOT   M00938	// R_REAR SAFETY SENSOR
AND NOT   M0093C	// RT_2D CODE TM OUT
AND NOT   M0093D	// RT_2D CODE NG
NOT
OR LOAD
LOAD      D080000.C	// ¡¤I¥ìu ALARM
AND       K00252	// LOADING ¡¾a ONLINE
OR LOAD
LOAD      D080400.C	// ¨ú©£¡¤I¥ìu ALARM
AND       K00253	// UNLOADING ¡¾a ONLINE
OR LOAD
OR NOT    M01233	// SYSTEM RIGHT LEFT
OUT       M01235	// RIGHT ALARM
; L773
LOAD NOT  M01235	// RIGHT ALARM
OUT       M01231	// R.ERR:0    R.GOOD:1

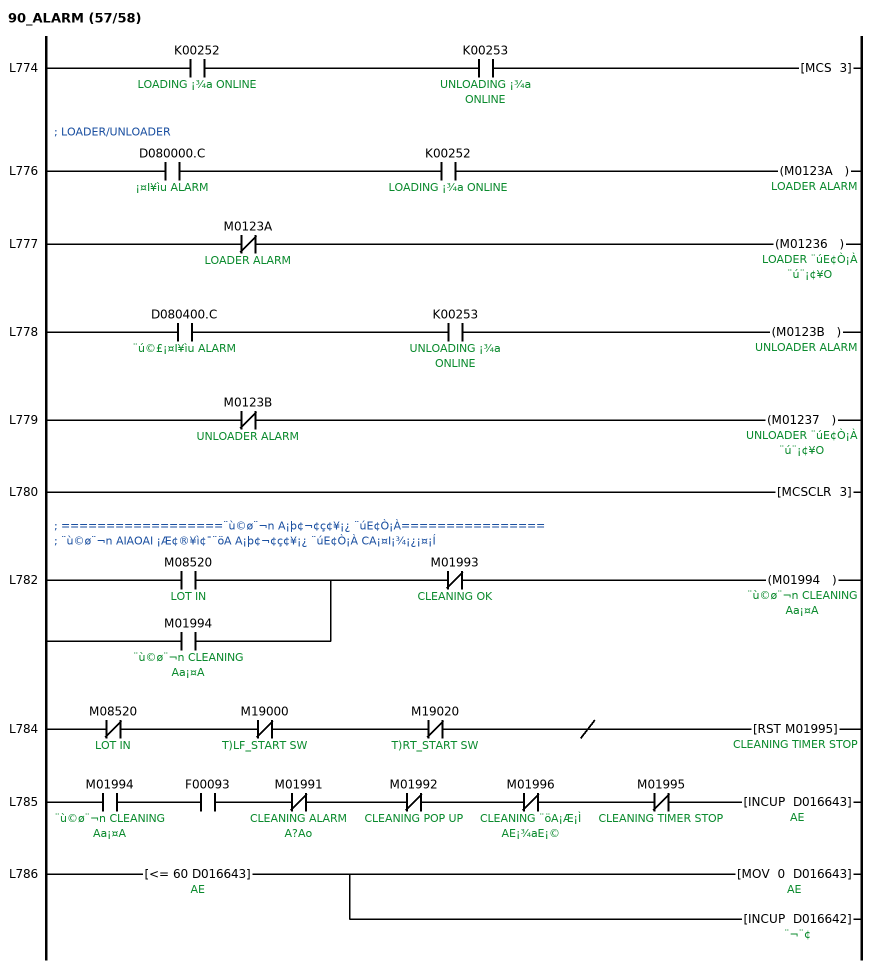
; L774
LOAD      K00252	// LOADING ¡¾a ONLINE
AND       K00253	// UNLOADING ¡¾a ONLINE
MCS       3
// LOADER/UNLOADER
; L776
LOAD      D080000.C	// ¡¤I¥ìu ALARM
AND       K00252	// LOADING ¡¾a ONLINE
OUT       M0123A	// LOADER ALARM
; L777
LOAD NOT  M0123A	// LOADER ALARM
OUT       M01236	// LOADER ¨úE¢Ò¡À ¨ú¨¡¢¥O
; L778
LOAD      D080400.C	// ¨ú©£¡¤I¥ìu ALARM
AND       K00253	// UNLOADING ¡¾a ONLINE
OUT       M0123B	// UNLOADER ALARM
; L779
LOAD NOT  M0123B	// UNLOADER ALARM
OUT       M01237	// UNLOADER ¨úE¢Ò¡À ¨ú¨¡¢¥O
; L780
MCSCLR    3
// ==================¨ù©ø¨¬n A¡þ¢¬¢ç¢¥¡¿ ¨úE¢Ò¡À================
; L782
LOAD      M08520	// LOT IN
OR        M01994	// ¨ù©ø¨¬n CLEANING Aa¡¤A
AND NOT   M01993	// CLEANING OK
OUT       M01994	// ¨ù©ø¨¬n CLEANING Aa¡¤A
// output comment: ¨ù©ø¨¬n AIAOAI ¡Æ¢®¥ì¢¯¨öA A¡þ¢¬¢ç¢¥¡¿ ¨úE¢Ò¡À CA¡¤I¡¾¡¿¡¤¡Í
; L784
LOAD NOT  M08520	// LOT IN
AND NOT   M19000	// T)LF_START SW
AND NOT   M19020	// T)RT_START SW
NOT
RST       M01995	// CLEANING TIMER STOP
; L785
LOAD      M01994	// ¨ù©ø¨¬n CLEANING Aa¡¤A
AND       F00093
AND NOT   M01991	// CLEANING ALARM A?Ao
AND NOT   M01992	// CLEANING POP UP
AND NOT   M01996	// CLEANING ¨öA¡Æ¡Ì AE¡¾aE¡©
AND NOT   M01995	// CLEANING TIMER STOP
INCUP     D016643	// AE
; L786
LOAD<=    60 D016643	// AE
MOV       0 D016643	// AE
INCUP     D016642	// ¨¬¨¢

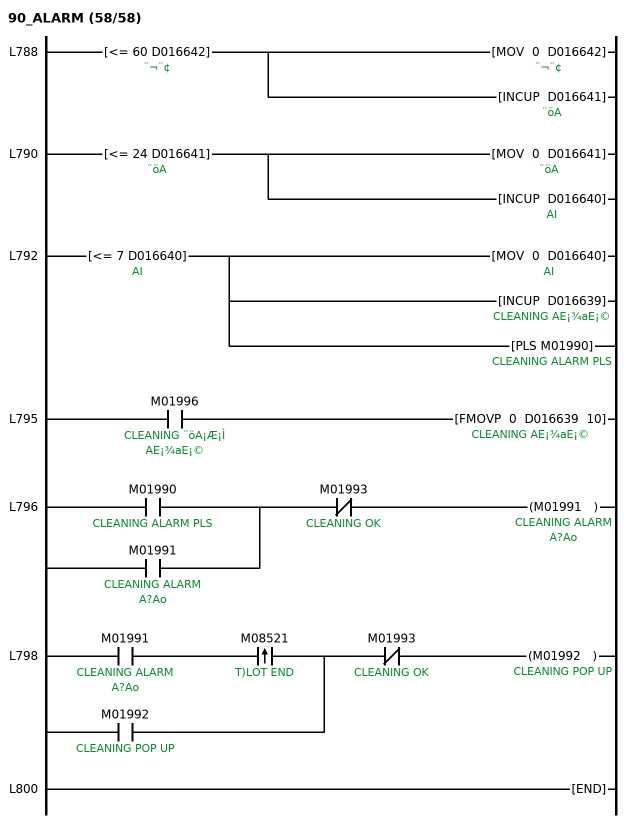
; L788
LOAD<=    60 D016642	// ¨¬¨¢
MOV       0 D016642	// ¨¬¨¢
INCUP     D016641	// ¨öA
; L790
LOAD<=    24 D016641	// ¨öA
MOV       0 D016641	// ¨öA
INCUP     D016640	// AI
; L792
LOAD<=    7 D016640	// AI
MOV       0 D016640	// AI
INCUP     D016639	// CLEANING AE¡¾aE¡©
OUTP      M01990	// CLEANING ALARM PLS
; L795
LOAD      M01996	// CLEANING ¨öA¡Æ¡Ì AE¡¾aE¡©
FMOVP     0 D016639 10	// CLEANING AE¡¾aE¡©
; L796
LOAD      M01990	// CLEANING ALARM PLS
OR        M01991	// CLEANING ALARM A?Ao
AND NOT   M01993	// CLEANING OK
OUT       M01991	// CLEANING ALARM A?Ao
; L798
LOAD      M01991	// CLEANING ALARM A?Ao
ANDP      M08521	// T)LOT END
OR        M01992	// CLEANING POP UP
AND NOT   M01993	// CLEANING OK
OUT       M01992	// CLEANING POP UP
; L800
END

PROGRAM 91_DEVICE_CHANGE (task: ¨ö¨¬A¥ì CA¡¤I¡¾¡¿¡¤¡Í)

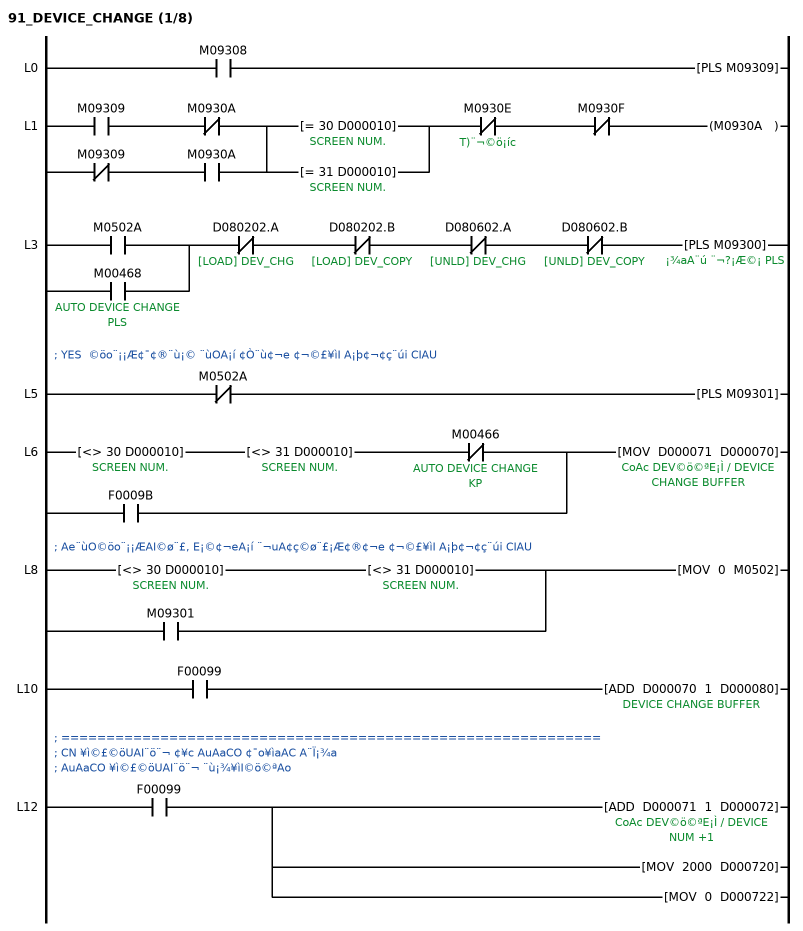
; L0
LOAD      M09308
OUTP      M09309
; L1
LOAD      M09309
AND NOT   M0930A
LOAD NOT  M09309
AND       M0930A
OR LOAD
LOAD=     30 D000010	// SCREEN NUM.
OR=       31 D000010	// SCREEN NUM.
AND LOAD
AND NOT   M0930E	// T)¨¬©ö¡íc
AND NOT   M0930F
OUT       M0930A
; L3
LOAD      M0502A
OR        M00468	// AUTO DEVICE CHANGE PLS
AND NOT   D080202.A	// [LOAD] DEV_CHG
AND NOT   D080202.B	// [LOAD] DEV_COPY
AND NOT   D080602.A	// [UNLD] DEV_CHG
AND NOT   D080602.B	// [UNLD] DEV_COPY
OUTP      M09300	// ¡¾aA¨ú ¨¬?¡Æ©¡ PLS
; L5
LOAD NOT  M0502A
OUTP      M09301
// output comment: YES  ©öo¨¡¡Æ¢¯¢®¨ù¡© ¨ùOA¡í ¢Ò¨ù¢¬e ¢¬©£¥ìI A¡þ¢¬¢ç¨úi CIAU
; L6
LOAD<>    30 D000010	// SCREEN NUM.
AND<>     31 D000010	// SCREEN NUM.
AND NOT   M00466	// AUTO DEVICE CHANGE KP
OR        F0009B
MOV       D000071 D000070	// CoAc DEV©ö©ªE¡Ì / DEVICE CHANGE BUFFER
; L8
LOAD<>    30 D000010	// SCREEN NUM.
AND<>     31 D000010	// SCREEN NUM.
OR        M09301
MOV       0 M0502
// output comment: Ae¨ùO©öo¨¡¡ÆAI©ø¨£, E¡©¢¬eA¡í ¨¬uA¢ç©ø¨£¡Æ¢®¢¬e ¢¬©£¥ìI A¡þ¢¬¢ç¨úi CIAU
; L10
LOAD      F00099
ADD       D000070 1 D000080	// DEVICE CHANGE BUFFER
// ============================================================
; L12
LOAD      F00099
ADD       D000071 1 D000072	// CoAc DEV©ö©ªE¡Ì / DEVICE NUM +1
MOV       2000 D000720
MOV       0 D000722
// output comment: CN ¥ì©£©öUAI¨ö¨¬ ¢¥c AuAaCO ¢¯o¥ìaAC A¨Ï¡¾a
// output comment: AuAaCO ¥ì©£©öUAI¨ö¨¬ ¨ù¡¾¥ìI©ö©ªAo

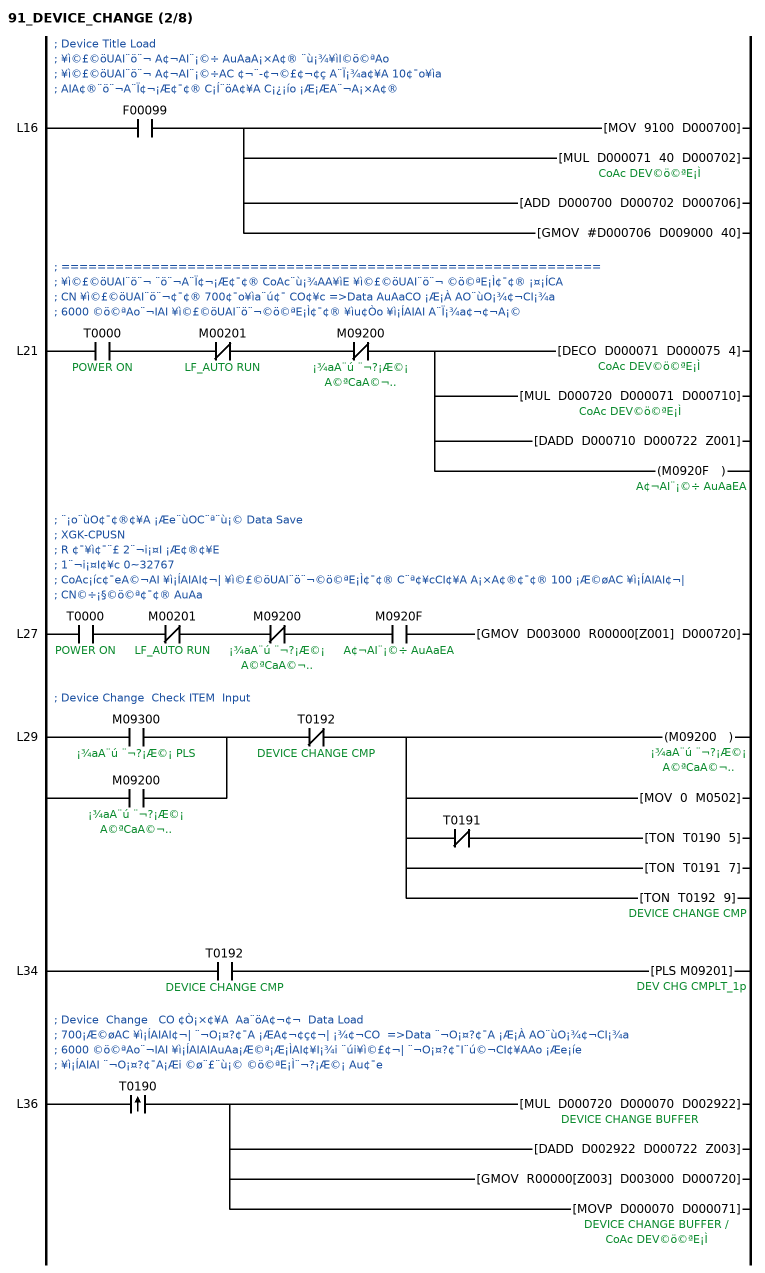
// Device Title Load
; L16
LOAD      F00099
MOV       9100 D000700
MUL       D000071 40 D000702	// CoAc DEV©ö©ªE¡Ì
ADD       D000700 D000702 D000706
GMOV      #D000706 D009000 40
// output comment: ¥ì©£©öUAI¨ö¨¬ A¢¬AI¨¡©÷ AuAaA¡×A¢® ¨ù¡¾¥ìI©ö©ªAo
// output comment: ¥ì©£©öUAI¨ö¨¬ A¢¬AI¨¡©÷AC ¢¬¨­¢¬©£¢¬¢ç A¨Ï¡¾a¢¥A 10¢¯o¥ìa
// output comment: AIA¢®¨ö¨¬A¨Ï¢¬¡Æ¢¯¢® C¡Í¨öA¢¥A C¡¿¡ío ¡Æ¡ÆA¨¬A¡×A¢®
// ============================================================
; L21
LOAD      T0000	// POWER ON
AND NOT   M00201	// LF_AUTO RUN
AND NOT   M09200	// ¡¾aA¨ú ¨¬?¡Æ©¡ A©ªCaA©¬..
DECO      D000071 D000075 4	// CoAc DEV©ö©ªE¡Ì
MUL       D000720 D000071 D000710	// CoAc DEV©ö©ªE¡Ì
DADD      D000710 D000722 Z001
OUT       M0920F	// A¢¬AI¨¡©÷ AuAaEA
// output comment: ¥ì©£©öUAI¨ö¨¬ ¨ö¨¬A¨Ï¢¬¡Æ¢¯¢® CoAc¨ù¡¾AA¥ìE ¥ì©£©öUAI¨ö¨¬ ©ö©ªE¡Ì¢¯¢® ¡¤¡ÍCA
// output comment: CN ¥ì©£©öUAI¨ö¨¬¢¯¢® 700¢¯o¥ìa¨ú¢¯ CO¢¥c =>Data AuAaCO ¡Æ¡À AO¨ùO¡¾¢¬CI¡¾a
// output comment: 6000 ©ö©ªAo¨¬IAI ¥ì©£©öUAI¨ö¨¬©ö©ªE¡Ì¢¯¢® ¥ìu¢Òo ¥ì¡ÍAIAI A¨Ï¡¾a¢¬¢¬A¡©
// ¨¡o¨ùO¢¯¢®¢¥A ¡Æe¨ùOC¨ª¨ù¡© Data Save
// XGK-CPUSN
// R ¢¯¥ì¢¯¨£ 2¨¬i¡¤I ¡Æ¢®¢¥E
// 1¨¬i¡¤I¢¥c 0~32767
; L27
LOAD      T0000	// POWER ON
AND NOT   M00201	// LF_AUTO RUN
AND NOT   M09200	// ¡¾aA¨ú ¨¬?¡Æ©¡ A©ªCaA©¬..
AND       M0920F	// A¢¬AI¨¡©÷ AuAaEA
GMOV      D003000 R00000[Z001] D000720
// output comment: CoAc¡íc¢¯eA©¬AI ¥ì¡ÍAIAI¢¬| ¥ì©£©öUAI¨ö¨¬©ö©ªE¡Ì¢¯¢® C¨ª¢¥cCI¢¥A A¡×A¢®¢¯¢® 100 ¡Æ©øAC ¥ì¡ÍAIAI¢¬| CN©÷¡§©ö©ª¢¯¢® AuAa
// Device Change  Check ITEM  Input
; L29
LOAD      M09300	// ¡¾aA¨ú ¨¬?¡Æ©¡ PLS
OR        M09200	// ¡¾aA¨ú ¨¬?¡Æ©¡ A©ªCaA©¬..
AND NOT   T0192	// DEVICE CHANGE CMP
OUT       M09200	// ¡¾aA¨ú ¨¬?¡Æ©¡ A©ªCaA©¬..
MOV       0 M0502
MPUSH
AND NOT   T0191
TON       T0190 5
MPOP
TON       T0191 7
TON       T0192 9	// DEVICE CHANGE CMP
; L34
LOAD      T0192	// DEVICE CHANGE CMP
OUTP      M09201	// DEV CHG CMPLT_1p
// Device  Change   CO ¢Ò¡×¢¥A  Aa¨öA¢¬¢¬  Data Load
; L36
LOADP     T0190
MUL       D000720 D000070 D002922	// DEVICE CHANGE BUFFER
DADD      D002922 D000722 Z003
GMOV      R00000[Z003] D003000 D000720
MOVP      D000070 D000071	// DEVICE CHANGE BUFFER / CoAc DEV©ö©ªE¡Ì
// output comment: 700¡Æ©øAC ¥ì¡ÍAIAI¢¬| ¨¬O¡¤?¢¯A ¡ÆA¢¬¢ç¢¬| ¡¾¢¬CO  =>Data ¨¬O¡¤?¢¯A ¡Æ¡À AO¨ùO¡¾¢¬CI¡¾a
// output comment: 6000 ©ö©ªAo¨¬IAI ¥ì¡ÍAIAIAuAa¡Æ©ª¡Æ¡ÌAI¢¥I¡¾i ¨úi¥ì©£¢¬| ¨¬O¡¤?¢¯I¨ú©¬CI¢¥AAo ¡Æe¡íe
// output comment: ¥ì¡ÍAIAI ¨¬O¡¤?¢¯A¡Æi ©ø¨£¨ù¡© ©ö©ªE¡Ì¨¬?¡Æ©¡ Au¢¯e

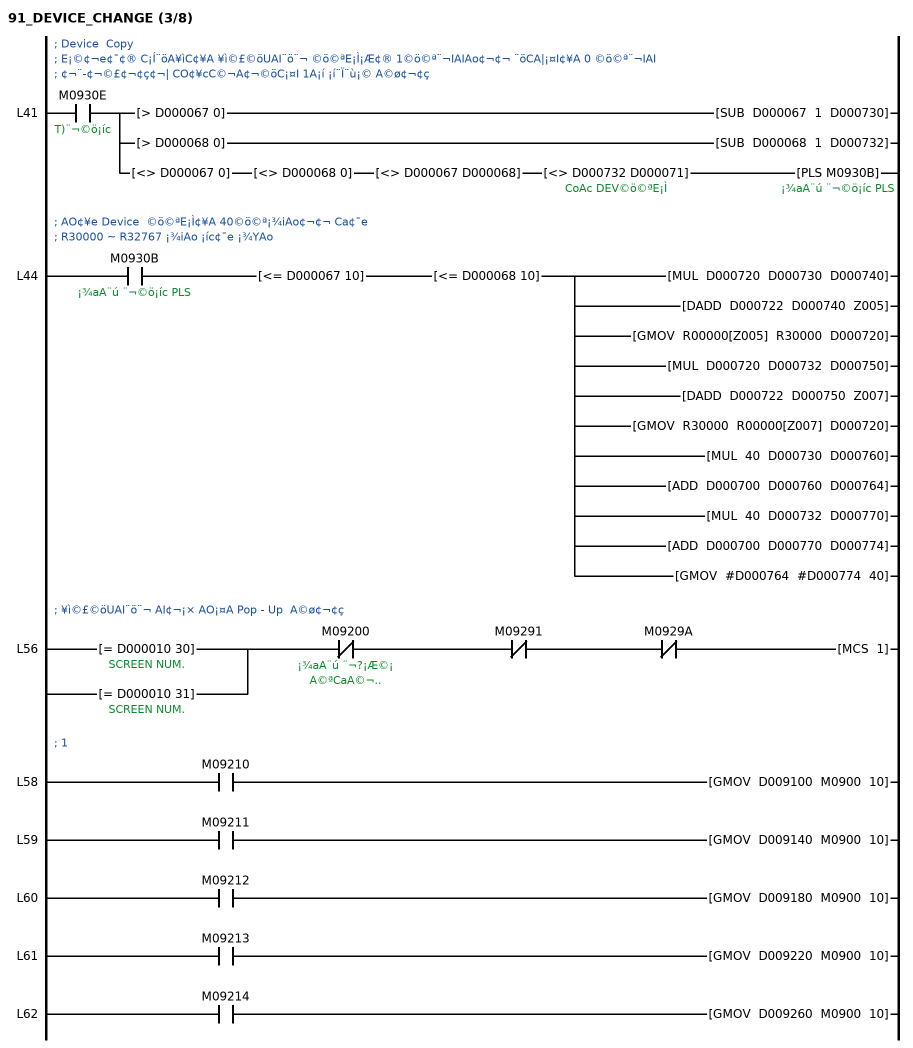
// Device  Copy
; L41
LOAD      M0930E	// T)¨¬©ö¡íc
MPUSH
AND>      D000067 0
SUB       D000067 1 D000730
MLOAD
AND>      D000068 0
SUB       D000068 1 D000732
MPOP
AND<>     D000067 0
AND<>     D000068 0
AND<>     D000067 D000068
AND<>     D000732 D000071	// CoAc DEV©ö©ªE¡Ì
OUTP      M0930B	// ¡¾aA¨ú ¨¬©ö¡íc PLS
// output comment: E¡©¢¬e¢¯¢® C¡Í¨öA¥ìC¢¥A ¥ì©£©öUAI¨ö¨¬ ©ö©ªE¡Ì¡Æ¢® 1©ö©ª¨¬IAIAo¢¬¢¬ ¨öCA|¡¤I¢¥A 0 ©ö©ª¨¬IAI
// output comment: ¢¬¨­¢¬©£¢¬¢ç¢¬| CO¢¥cC©¬A¢¬©öC¡¤I 1A¡í ¡í¨Ï¨ù¡© A©ø¢¬¢ç
; L44
LOAD      M0930B	// ¡¾aA¨ú ¨¬©ö¡íc PLS
AND<=     D000067 10
AND<=     D000068 10
MUL       D000720 D000730 D000740
DADD      D000722 D000740 Z005
GMOV      R00000[Z005] R30000 D000720
MUL       D000720 D000732 D000750
DADD      D000722 D000750 Z007
GMOV      R30000 R00000[Z007] D000720
MUL       40 D000730 D000760
ADD       D000700 D000760 D000764
MUL       40 D000732 D000770
ADD       D000700 D000770 D000774
GMOV      #D000764 #D000774 40
// output comment: AO¢¥e Device  ©ö©ªE¡Ì¢¥A 40©ö©ª¡¾iAo¢¬¢¬ Ca¢¯e
// output comment: R30000 ~ R32767 ¡¾iAo ¡íc¢¯e ¡¾YAo
// ¥ì©£©öUAI¨ö¨¬ AI¢¬¡× AO¡¤A Pop - Up  A©ø¢¬¢ç
; L56
LOAD=     D000010 30	// SCREEN NUM.
OR=       D000010 31	// SCREEN NUM.
AND NOT   M09200	// ¡¾aA¨ú ¨¬?¡Æ©¡ A©ªCaA©¬..
AND NOT   M09291
AND NOT   M0929A
MCS       1
; L58
LOAD      M09210
GMOV      D009100 M0900 10
// output comment: 1
; L59
LOAD      M09211
GMOV      D009140 M0900 10
; L60
LOAD      M09212
GMOV      D009180 M0900 10
; L61
LOAD      M09213
GMOV      D009220 M0900 10
; L62
LOAD      M09214
GMOV      D009260 M0900 10

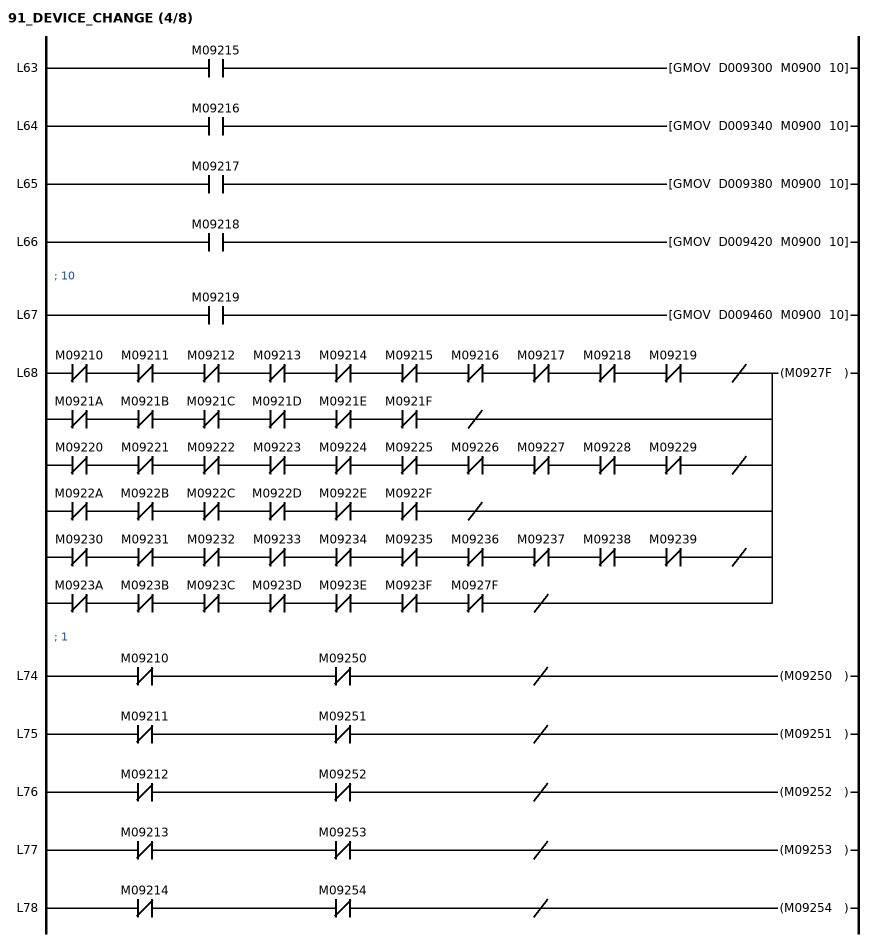
; L63
LOAD      M09215
GMOV      D009300 M0900 10
; L64
LOAD      M09216
GMOV      D009340 M0900 10
; L65
LOAD      M09217
GMOV      D009380 M0900 10
; L66
LOAD      M09218
GMOV      D009420 M0900 10
; L67
LOAD      M09219
GMOV      D009460 M0900 10
// output comment: 10
; L68
LOAD NOT  M09210
AND NOT   M09211
AND NOT   M09212
AND NOT   M09213
AND NOT   M09214
AND NOT   M09215
AND NOT   M09216
AND NOT   M09217
AND NOT   M09218
AND NOT   M09219
NOT
LOAD NOT  M0921A
AND NOT   M0921B
AND NOT   M0921C
AND NOT   M0921D
AND NOT   M0921E
AND NOT   M0921F
NOT
OR LOAD
LOAD NOT  M09220
AND NOT   M09221
AND NOT   M09222
AND NOT   M09223
AND NOT   M09224
AND NOT   M09225
AND NOT   M09226
AND NOT   M09227
AND NOT   M09228
AND NOT   M09229
NOT
OR LOAD
LOAD NOT  M0922A
AND NOT   M0922B
AND NOT   M0922C
AND NOT   M0922D
AND NOT   M0922E
AND NOT   M0922F
NOT
OR LOAD
LOAD NOT  M09230
AND NOT   M09231
AND NOT   M09232
AND NOT   M09233
AND NOT   M09234
AND NOT   M09235
AND NOT   M09236
AND NOT   M09237
AND NOT   M09238
AND NOT   M09239
NOT
OR LOAD
LOAD NOT  M0923A
AND NOT   M0923B
AND NOT   M0923C
AND NOT   M0923D
AND NOT   M0923E
AND NOT   M0923F
AND NOT   M0927F
NOT
OR LOAD
OUT       M0927F
; L74
LOAD NOT  M09210
AND NOT   M09250
NOT
OUT       M09250
// output comment: 1
; L75
LOAD NOT  M09211
AND NOT   M09251
NOT
OUT       M09251
; L76
LOAD NOT  M09212
AND NOT   M09252
NOT
OUT       M09252
; L77
LOAD NOT  M09213
AND NOT   M09253
NOT
OUT       M09253
; L78
LOAD NOT  M09214
AND NOT   M09254
NOT
OUT       M09254

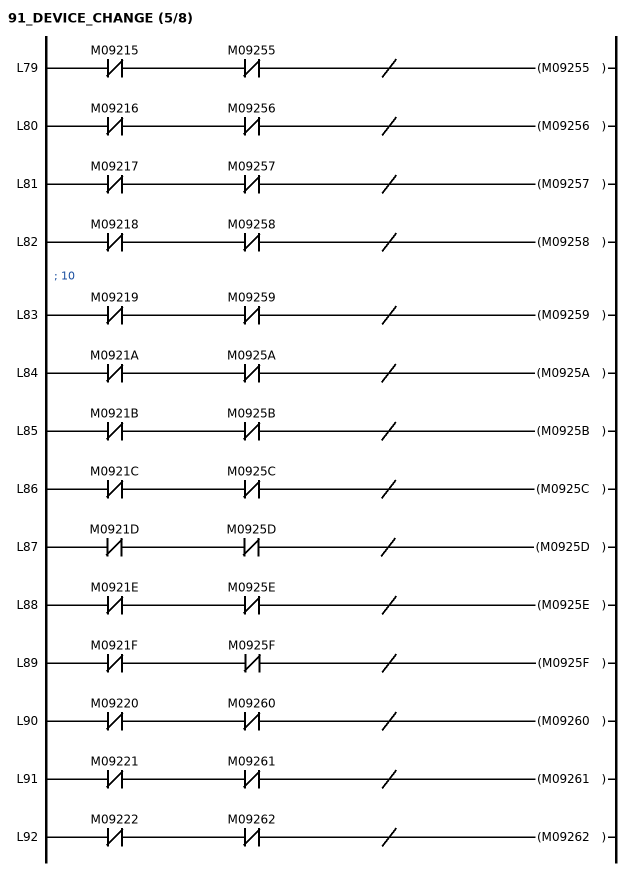
; L79
LOAD NOT  M09215
AND NOT   M09255
NOT
OUT       M09255
; L80
LOAD NOT  M09216
AND NOT   M09256
NOT
OUT       M09256
; L81
LOAD NOT  M09217
AND NOT   M09257
NOT
OUT       M09257
; L82
LOAD NOT  M09218
AND NOT   M09258
NOT
OUT       M09258
; L83
LOAD NOT  M09219
AND NOT   M09259
NOT
OUT       M09259
// output comment: 10
; L84
LOAD NOT  M0921A
AND NOT   M0925A
NOT
OUT       M0925A
; L85
LOAD NOT  M0921B
AND NOT   M0925B
NOT
OUT       M0925B
; L86
LOAD NOT  M0921C
AND NOT   M0925C
NOT
OUT       M0925C
; L87
LOAD NOT  M0921D
AND NOT   M0925D
NOT
OUT       M0925D
; L88
LOAD NOT  M0921E
AND NOT   M0925E
NOT
OUT       M0925E
; L89
LOAD NOT  M0921F
AND NOT   M0925F
NOT
OUT       M0925F
; L90
LOAD NOT  M09220
AND NOT   M09260
NOT
OUT       M09260
; L91
LOAD NOT  M09221
AND NOT   M09261
NOT
OUT       M09261
; L92
LOAD NOT  M09222
AND NOT   M09262
NOT
OUT       M09262

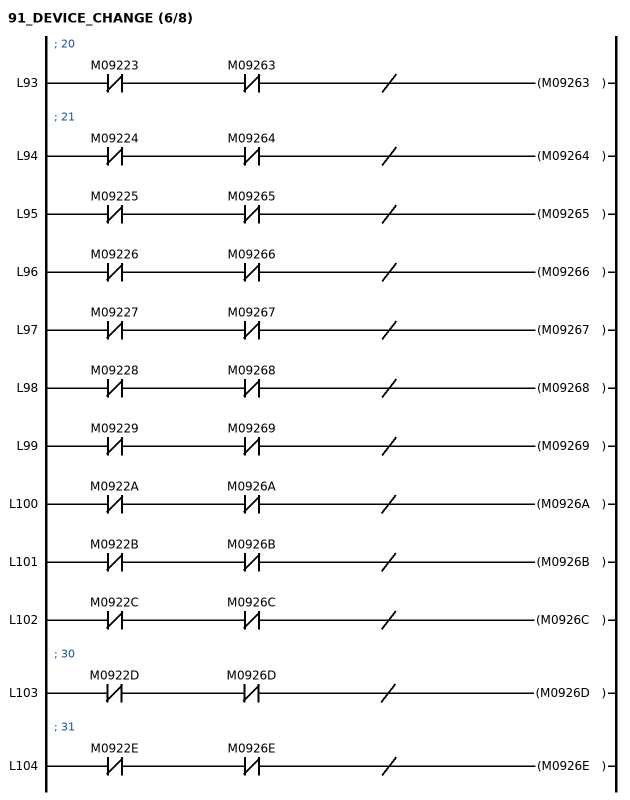
; L93
LOAD NOT  M09223
AND NOT   M09263
NOT
OUT       M09263
// output comment: 20
; L94
LOAD NOT  M09224
AND NOT   M09264
NOT
OUT       M09264
// output comment: 21
; L95
LOAD NOT  M09225
AND NOT   M09265
NOT
OUT       M09265
; L96
LOAD NOT  M09226
AND NOT   M09266
NOT
OUT       M09266
; L97
LOAD NOT  M09227
AND NOT   M09267
NOT
OUT       M09267
; L98
LOAD NOT  M09228
AND NOT   M09268
NOT
OUT       M09268
; L99
LOAD NOT  M09229
AND NOT   M09269
NOT
OUT       M09269
; L100
LOAD NOT  M0922A
AND NOT   M0926A
NOT
OUT       M0926A
; L101
LOAD NOT  M0922B
AND NOT   M0926B
NOT
OUT       M0926B
; L102
LOAD NOT  M0922C
AND NOT   M0926C
NOT
OUT       M0926C
; L103
LOAD NOT  M0922D
AND NOT   M0926D
NOT
OUT       M0926D
// output comment: 30
; L104
LOAD NOT  M0922E
AND NOT   M0926E
NOT
OUT       M0926E
// output comment: 31

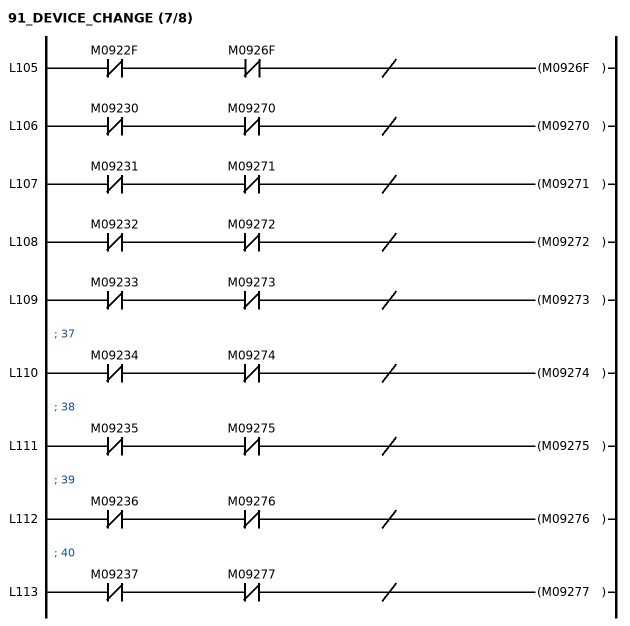
; L105
LOAD NOT  M0922F
AND NOT   M0926F
NOT
OUT       M0926F
; L106
LOAD NOT  M09230
AND NOT   M09270
NOT
OUT       M09270
; L107
LOAD NOT  M09231
AND NOT   M09271
NOT
OUT       M09271
; L108
LOAD NOT  M09232
AND NOT   M09272
NOT
OUT       M09272
; L109
LOAD NOT  M09233
AND NOT   M09273
NOT
OUT       M09273
; L110
LOAD NOT  M09234
AND NOT   M09274
NOT
OUT       M09274
// output comment: 37
; L111
LOAD NOT  M09235
AND NOT   M09275
NOT
OUT       M09275
// output comment: 38
; L112
LOAD NOT  M09236
AND NOT   M09276
NOT
OUT       M09276
// output comment: 39
; L113
LOAD NOT  M09237
AND NOT   M09277
NOT
OUT       M09277
// output comment: 40

